(* PLC project test, Неизвестно Unnamed 1 *)
(* stored: creationDateTime 2025-01-15T16:56:00, modificationDateTime 2025-01-16T04:38:44 *)

TYPE TError : (E_SUCCESS, E_ID, E_HEAD, E_INDEX, E_ITEMPOS, E_ITEM, E_GRID, E_AXIS, E_PRIO, E_MATER, E_PROFILE, E_VALUE, E_STACKSIZE, E_ROOT, E_ITEMSIZE, E_STEPSIZE, E_TIMESIZE, E_NOTREADY, E_STRUCT, E_VALIDATE, E_LOC2ABS, E_ABS2LOC, E_GETTEMP, E_SETTEMP, E_CHECKVALID, E_LINKITEMS, E_PROCESS, E_PREPROC, E_POSTPROC, E_BADTEMP, E_STATE, E_CHECK, E_FAIL, W_PERIOD) := E_SUCCESS;
END_TYPE

TYPE TStat : STRUCT
  RDY : BOOL := TRUE;
  DBG : BOOL := TRUE;
  ERR : TError := E_SUCCESS;
  PAR : UINT := 0;
  STR : STRING := '';
END_STRUCT;
END_TYPE

TYPE LOGLEVEL : (CRITICAL, WARNING, INFO, DEBUG) := DEBUG;
END_TYPE

(* Приоритет по коду ошибки *)
FUNCTION Err2Lev : LOGLEVEL
  VAR_INPUT
    Err : TError := E_SUCCESS;  (* Флаг ошибки *)
  END_VAR

            CASE Err OF
E_SUCCESS:  
  Err2Lev:=INFO;  
W_PERIOD:   
  Err2Lev:=WARNING;  
ELSE        
  Err2Lev:=CRITICAL;  
END_CASE;
RETURN;
          
END_FUNCTION

(* Выдает строку по коду ошибки *)
FUNCTION MakeMsg : STRING
  VAR_INPUT
    S0 : STRING := '';  (* Строка 0 *)
    S1 : STRING := '';  (* Строка 1 *)
    S2 : STRING := '';  (* Строка 2 *)
    S3 : STRING := '';  (* Строка 3 *)
  END_VAR
  VAR
    BLOG : BOOL := FALSE;  (* Флаг работы *)
  END_VAR

            {{ BLOG = __GET_GLOBAL_STAT()->DBG; }}
if (BLOG) then 
  MakeMsg:=concat(concat(concat(S0, S1), S2), S3); 
else 
  MakeMsg:=''; 
end_if;
          
END_FUNCTION

(* Выдает строку по коду ошибки *)
FUNCTION Err2Str : STRING
  VAR_INPUT
    ERR : TError := E_SUCCESS;  (* Код ошибки *)
  END_VAR

            case ERR of
(* Информационные сообщения *)
E_SUCCESS:      Err2Str := 'Succeeded!';

(* Критические ошибки *)
E_FAIL:         Err2Str := 'Unexpected error';
E_STATE:        Err2Str := 'Program state error';
E_CHECK:        Err2Str := 'Check point error';
E_HEAD:         Err2Str := 'Invalid head';
E_INDEX:        Err2Str := 'Invalid index';
E_ITEMPOS:      Err2Str := 'Invalid item position';
E_ITEM:         Err2Str := 'Invalid element';
E_GRID:         Err2Str := 'Invalid grid';
E_AXIS:         Err2Str := 'Invalid axis';
E_PRIO:         Err2Str := 'Invalid prio';
E_MATER:        Err2Str := 'Invalid mater';
E_PROFILE:      Err2Str := 'Invalid profile';
E_VALUE:        Err2Str := 'Invalid value';
E_ROOT:         Err2Str := 'Invalid ROOT';
E_ITEMSIZE:     Err2Str := 'Bad ItemAt size';
E_STEPSIZE:     Err2Str := 'Bad axis step';
E_TIMESIZE:     Err2Str := 'Bad time step';
E_STACKSIZE:    Err2Str := 'Small stacksize';
E_NOTREADY:     Err2Str := 'Object dont ready';
E_LOC2ABS:      Err2Str := 'Loc2Abs error';
E_ABS2LOC:      Err2Str := 'Abs2Loc error';
E_VALIDATE:     Err2Str := 'Validate error';
E_CHECKVALID:   Err2Str := 'CheckValid error';
E_LINKITEMS:    Err2Str := 'LinkItems error';
E_PROCESS:      Err2Str := 'Process item error';
E_BADTEMP:      Err2Str := 'GetTemp error';

(* Предупреждения *)
W_PERIOD:       Err2Str := 'Small period';
else            Err2Str := 'Unknown error';
end_case;

          
END_FUNCTION

(* Протоколирование ошибки *)
FUNCTION LogMsg : STRING
  VAR_INPUT
    STR : STRING := '';  (* Строка для протокола *)
    LVL : LOGLEVEL := DEBUG;  (* Уровень сообщения (по умолчанию - Debug) *)
    ERR : TError := E_SUCCESS;  (* Код ошибки *)
  END_VAR

            {{
  #ifdef _BEREMIZ_H_
    #define __LOG_MSG(level,string,length) LogMessage(level,(char *)string,length)
  #else
    #define __LOG_MSG(level,string,length) printf("%s\n", (char *)string)
  #endif
  TSTAT *pStat = __GET_GLOBAL_STAT();
  if (LVL!=LOGLEVEL__DEBUG || (LVL==LOGLEVEL__DEBUG && pStat->DBG)) {
    if (STR.len) __LOG_MSG(LVL, (char *)STR.body, STR.len);
  }
  if (ERR!=TERROR__E_SUCCESS) {
    pStat->ERR=ERR;
    LVL=ERR2LEV(1,NULL,ERR); 
    STR=ERR2STR(1,NULL,ERR);
    if (STR.len) __LOG_MSG(LVL,(char *)STR.body,STR.len);
  }
  return (LOGMSG = __INIT_STRING);
}}

          
END_FUNCTION

PROGRAM Test
  VAR
    LocalVar0 : DINT;
  END_VAR

            
LocalVar0 := 1;

          
END_PROGRAM

PROGRAM Simulation
  VAR
    T1 : TON;
    P_Cooling : TIME := TIME#500ms;
    xReduceTemp : BOOL;
    T2 : TON;
    P_Environment : TIME := TIME#2s0ms;
    P_EnvironmentDoorOpen : TIME := TIME#1s0ms;
    xRaiseTemp : BOOL;
    timTemp : TIME;
    iCounter : INT;
  END_VAR

            iCounter:=0;
(*
    IF Glob_VAR.bCompressor THEN
      T1(IN:= Glob_Var.bCompressor, PT:= P_Cooling, Q=&gt;xReduceTemp);
    
      IF xReduceTemp THEN
        Glob_Var.rTempActual := Glob_Var.rTempActual-0.1;
        T1(IN:=FALSE);
      END_IF
    END_IF

    timTemp:=SEL(Glob_Var.rDoorOpen, P_Environment, P_EnvironmentDoorOpen);

    T2(IN:= TRUE, PT:= timTemp, Q=&gt;xRaiseTemp);
    
    IF xRaiseTemp THEN
      Glob_Var.rTempActual := Glob_Var.rTempActual + 0.1;
      T2(IN:=FALSE);
    END_IF
*)

          
END_PROGRAM

CONFIGURATION Config0
  VAR_GLOBAL
    STAT : TStat;  (* Статус контроллера *)
  END_VAR
  RESOURCE Res0 ON PLC
    VAR_GLOBAL
      rTempActual : REAL := 8;
      rTempSet : REAL := 8;
      rDoorOpen : BOOL := FALSE;
      timAlarmThreshold : TIME := TIME#30ms;
      rDoorOpenThreshold : TIME := TIME#10s0ms;
      bCompressor : BOOL := false;
      bSignal : BOOL := FALSE;
      bLamp : BOOL := FALSE;
    END_VAR
    TASK MainTask(INTERVAL := T#20ms, PRIORITY := 0);
    PROGRAM Prog1 WITH MainTask : Simulation;
    PROGRAM Prog2 WITH MainTask : Test;
  END_RESOURCE
END_CONFIGURATION
